# B&R Automation Studio project BottleFiller (part 2)

#### Main.st
```iecst
PROGRAM _INIT
	(* Insert code here *)
	//Conveyor parameters
	MpAxisConvParType.AutoTune.Mode:=mcAXIS_TUNE_AUTOMATIC;
	MpAxisConvParType.AutoTune.MaxCurrentPercent:=80;
	MpAxisConvParType.AutoTune.MaxDistance:=30;
	MpAxisConvParType.AutoTune.MaxPositionError:=30;
	//Nozzle parameters
	MpAxisNozzleParType := MpAxisConvParType;
	MpAxisNozzleParType.Homing.Position:=195;
	//Cart parameters
	MpAxisCartParType := MpAxisConvParType;

	camNozzleParameters.CamSequence.Get.GetOnEnable:=1;
	camNozzleParameters.CamSequence.Get.Command:=mcGET_PAR_ACTUAL;
	camNozzleParameters.CamSequence.Data.DataAddress:=ADR(configCamNozzle);
	camNozzleParameters.CamSequence.Data.DataSize:=SIZEOF(configCamNozzle);
	camNozzleParameters.CamSequence.Set.Command:=mcSET_UPDATE_FROM_ADR;
	camNozzleParameters.CamSequence.Set.Mode:=mcAXIS_CAM_SEQ_SET_ON_UPDATE;
END_PROGRAM

PROGRAM _CYCLIC
	(* Insert code here *)
	//axis declaration
	MpAxisConv(MpLink := ADR(axisConv), Enable := 1, Parameters := ADR(MpAxisConvParType), AutoTune := 1);
	MpAxisCart(MpLink := ADR(axisCart), Enable := 1, Parameters := ADR(MpAxisCartParType),   AutoTune := 1);
	MpAxisNozzle(MpLink := ADR(axisNozzle), Enable := 1, Parameters := ADR(MpAxisNozzleParType),  AutoTune := 1);

	//sequence parameters
	configCamNozzle.State[3].CamID:=STRING_TO_USINT(gControl.currentBottleType);

	//Sequence declaration
	camSeq(MpLink := ADR(axisCart), Enable := 1, Parameters := ADR(camParameters), MpLinkMaster := ADR(axisConv));
	camSeqNozzle(MpLink := ADR(axisNozzle), Enable := 1, Parameters := ADR(camNozzleParameters), MpLinkMaster := ADR(axisConv));

	//conveyor management
	MpAxisConvParType.Velocity:=gAxisUpdate.Conveyor.Velocity;
	MpAxisConv.ErrorReset:=gControl.Conveyor.errorReset;
	MpAxisConv.Power:=gControl.power;
	MpAxisConv.Home:=gControl.Conveyor.home;
	MpAxisConv.Stop:=gControl.Conveyor.stop;
	MpAxisConv.JogNegative:=gControl.Conveyor.jogNegative;
	MpAxisConv.JogPositive:=gControl.Conveyor.jogPositive;

	//Cart management
	MpAxisCart.ErrorReset:=gControl.Cart.errorReset;
	MpAxisCart.Power:=gControl.power;
	MpAxisCart.Home:=gControl.Cart.home;
	MpAxisCart.Stop:=gControl.Cart.stop;
	MpAxisCart.JogNegative:=gControl.Cart.jogNegative;
	MpAxisCart.JogPositive:=gControl.Cart.jogPositive;

	//nozzle Management
	MpAxisNozzle.ErrorReset:=gControl.Nozzle.errorReset;
	MpAxisNozzle.Power:=gControl.power;
	MpAxisNozzle.Home:=gControl.Nozzle.home;
	MpAxisNozzle.Stop:=gControl.Nozzle.stop;
	MpAxisNozzle.JogNegative:=gControl.Nozzle.jogNegative;
	MpAxisNozzle.JogPositive:=gControl.Nozzle.jogPositive;

	//cam params
//	camSeq.Signal1:=gCamSeqParam.cart.signal1;
	camSeqNozzle.Signal1:=gCamSeqParam.nozzle.signal1;

	IF camSeqNozzle.UpdateDone THEN
		camSeqNozzle.Update:=0;
	END_IF;
	IF MpAxisConv.UpdateDone THEN
		MpAxisConv.Update:=0;
	END_IF;
	IF MpAxisNozzle.UpdateDone THEN
		MpAxisNozzle.Update:=0;
	END_IF;
	IF MpAxisCart.UpdateDone THEN
		MpAxisCart.Update:=0;
	END_IF;

	IF gControl.needUpdate THEN

		//conveyor
		MpAxisConvParType.Velocity:=STRING_TO_UINT(gAxisUpdate.staticVelocity);
		MpAxisConvParType.Jog.LimitPosition.FirstPosition:=gAxisUpdate.Conveyor.FirstPosition;
		MpAxisConvParType.Jog.LimitPosition.LastPosition:=gAxisUpdate.Conveyor.LastPosition;
		MpAxisConvParType.Position:=gAxisUpdate.Conveyor.Position;
		//MpAxisConvParType.Homing.Mode:=gAxisUpdate.Conveyor.Homing;
		//MpAxisConvParType.Velocity:=gAxisUpdate.Conveyor.Velocity;
		MpAxisConvParType.Jog.Velocity:=gAxisUpdate.Conveyor.Velocity;

		//cart
		MpAxisCartParType.Jog.LimitPosition.FirstPosition:=gAxisUpdate.Cart.FirstPosition;
		MpAxisCartParType.Jog.LimitPosition.LastPosition:=gAxisUpdate.Cart.LastPosition;
		MpAxisCartParType.Position:=gAxisUpdate.Cart.Position;
		//	MpAxisCartParType.Homing.Mode:=gAxisUpdate.Cart.Homing;
		MpAxisCartParType.Jog.Velocity:=50;

		//nozzle
		MpAxisNozzleParType.Jog.LimitPosition.FirstPosition:=gAxisUpdate.Nozzle.FirstPosition;
		MpAxisNozzleParType.Jog.LimitPosition.LastPosition:=gAxisUpdate.Nozzle.LastPosition;
		MpAxisNozzleParType.Position:=gAxisUpdate.Nozzle.Position;
		//	MpAxisNozzleParType.Homing.Mode:=gAxisUpdate.Nozzle.Homing;
		MpAxisNozzleParType.Jog.Velocity:=50;

		MpAxisNozzle.Update:=1;
		MpAxisConv.Update:=1;
		MpAxisCart.Update:=1;

		IF MpAxisNozzle.UpdateDone THEN
			MpAxisNozzle.Update:=0;
		END_IF;
		IF MpAxisCart.UpdateDone THEN
			MpAxisCart.Update:=0;
		END_IF;
		IF MpAxisConv.UpdateDone THEN
			MpAxisConv.Update:=0;
		END_IF;
		gControl.needUpdate:=0;
	END_IF;

	CASE gAxisCase OF
		HOLDON:
			IF NOT (MpAxisCart.Stopped AND MpAxisConv.Stopped AND MpAxisNozzle.Stopped)  THEN
				MpAxisCart.Stop:=1;
				MpAxisConv.Stop:=1;
				MpAxisNozzle.Stop:=1;
			END_IF;

			IF  MpAxisConv.Info.PLCopenState = mcAXIS_STANDSTILL AND MpAxisCart.Info.PLCopenState = mcAXIS_STANDSTILL AND MpAxisNozzle.Info.PLCopenState = mcAXIS_STANDSTILL THEN
				MpAxisCart.Stop:=0;
				MpAxisConv.Stop:=0;
				MpAxisNozzle.Stop:=0;
				gMainAction.stopped:=1;
			END_IF;

		POWERED:
			IF (gControl.power AND NOT gControl.stop AND NOT gAxisOutputs.Conveyor.error) THEN //error
				//power on axis
				MpAxisCart.Power:=1;
				MpAxisConv.Power:=1;
				MpAxisNozzle.Power:=1;

				IF MpAxisCart.PowerOn AND MpAxisConv.PowerOn AND MpAxisNozzle.PowerOn THEN
					gMainAction.powered:=1;
				END_IF;

			END_IF;

		HOMING:
			gControl.bottleCnt:=0;
			MpAxisCart.Home:=1;
			MpAxisConv.Home:=1;
			MpAxisNozzle.Home:=1;
			gMainAction.homed:=1;

		STANDSTILL:
			IF gControl.start THEN
				IF gControl.manual THEN
					gAxisCase:=onMOVE;
				ELSE
					gAxisCase:=CONNECT;
				END_IF;
			END_IF;

		CONNECT:
			MpAxisCart.Home:=0;
			MpAxisConv.Home:=0;
			MpAxisNozzle.Home:=0;
			camSeq.EndSequence:=0;
			camSeqNozzle.EndSequence:=0;
			camSeq.ErrorReset:=0;
			camSeq.StartSequence:=1;
			camSeqNozzle.StartSequence:=1;

			IF camSeq.Error THEN
				camSeq.ErrorReset:=1;
				camSeq.StartSequence:=0;
			END_IF;

			IF camSeq.InCam AND camSeqNozzle.InCam THEN
				camSeq.Signal1:=1;
				gMainAction.connected:=1;
				connectHelper:=0;
			END_IF;

		DISCONNECT:
			MpAxisCart.Home:=0;
			MpAxisConv.Home:=0;
			MpAxisNozzle.Home:=0;
			gMainAction.connected:=0;
			MpAxisConv.MoveVelocity:=0;
			camSeq.Signal1:=0;
			camSeqNozzle.Signal1:=0;
			camSeq.StartSequence:=0;
			camSeq.EndSequence:=1;
			camSeqNozzle.StartSequence:=0;
			camSeqNozzle.EndSequence:=1;
			IF NOT (camSeq.Running AND camSeqNozzle.Running) THEN
				gMainAction.disconnected:=1;
			END_IF;

		onMOVE:
			//karetka
			IF mouseEvent THEN
				IF gControl.Cart.safeLevelStop THEN
					gControl.Cart.stop:=gControl.Cart.safeLevelStop;
					IF MpAxisCartParType.Direction = 1 AND MpAxisCart.Position >= gControl.Cart.upperLimit THEN
						gControl.Cart.safeLevelStop:=0;
						gControl.Cart.stop:=0;
					ELSIF MpAxisCartParType.Direction = 0 AND MpAxisCart.Position <= gControl.Cart.lowerLimit THEN
						gControl.Cart.safeLevelStop:=0;
						gControl.Cart.stop:=0;
					END_IF;
				END_IF;

				IF gControl.Nozzle.safeLevelStop THEN
					gControl.Nozzle.stop:=gControl.Nozzle.safeLevelStop;
					IF MpAxisNozzleParType.Direction = 1 AND MpAxisNozzle.Position >= gControl.Nozzle.upperLimit THEN
						gControl.Nozzle.safeLevelStop:=0;
						gControl.Nozzle.stop:=0;
					ELSIF MpAxisNozzleParType.Direction = 0 AND MpAxisNozzle.Position <= gControl.Nozzle.lowerLimit THEN
						gControl.Nozzle.safeLevelStop:=0;
						gControl.Nozzle.stop:=0;
					END_IF;
				END_IF;

				MpAxisConv.MoveVelocity:=gControl.moveVelocity;

				IF gControl.Cart.onlyRight AND MpAxisCartParType.Direction = 0 THEN
					gControl.Cart.stop:=0;
					MpAxisCart.MoveVelocity:=gControl.Cart.moveVelocity;
				END_IF;

				IF gControl.Cart.onlyLeft AND MpAxisCartParType.Direction = 1 THEN
					gControl.Cart.stop:=0;
					MpAxisCart.MoveVelocity:=gControl.Cart.moveVelocity;
				END_IF;

				IF NOT gControl.Cart.onlyLeft AND NOT gControl.Cart.onlyRight THEN
					MpAxisCart.MoveVelocity:= NOT gControl.Cart.safeLevelStop AND gControl.Cart.moveVelocity;
				END_IF;

				//nozzle
				IF gControl.Nozzle.onlyRight AND MpAxisNozzleParType.Direction = 0 THEN
					gControl.Nozzle.stop:=0;
					MpAxisNozzle.MoveVelocity:=gControl.Nozzle.moveVelocity;
				END_IF;

				IF gControl.Nozzle.onlyLeft AND MpAxisNozzleParType.Direction = 1 THEN
					gControl.Nozzle.stop:=0;
					MpAxisNozzle.MoveVelocity:=gControl.Nozzle.moveVelocity;
				END_IF;

				IF NOT gControl.Nozzle.onlyLeft AND NOT gControl.Nozzle.onlyRight THEN
					MpAxisNozzle.MoveVelocity:= NOT gControl.Nozzle.safeLevelStop AND gControl.Nozzle.moveVelocity;
				END_IF;
			ELSE
				MpAxisConv.MoveVelocity:=gControl.moveVelocity;
				MpAxisConv.JogNegative:=gControl.Conveyor.jogNegative;
				MpAxisConv.JogPositive:=gControl.Conveyor.jogPositive;
				MpAxisCart.JogNegative:=gControl.Cart.jogNegative;
				MpAxisCart.JogPositive:=gControl.Cart.jogPositive;
				MpAxisNozzle.JogNegative:=gControl.Nozzle.jogNegative;
				MpAxisNozzle.JogPositive:=gControl.Nozzle.jogPositive;
			END_IF;
			IF MpAxisConv.Position > 0 THEN
				gMainAction.homed:=0;
			END_IF;

	END_CASE;

	controlInfo.Conveyor.error:=MpAxisConv.Error;
	controlInfo.Conveyor.isHomed:=MpAxisConv.IsHomed;
	controlInfo.Conveyor.isPowered:=MpAxisConv.PowerOn;
	controlInfo.Conveyor.position:=LREAL_TO_REAL(MpAxisConv.Position);
	controlInfo.Conveyor.velocity:=MpAxisConv.Velocity;
	controlInfo.Conveyor.updateDone:=MpAxisConv.UpdateDone;
	controlInfo.Conveyor.MoveActive:=MpAxisConv.Info.Jogging;

	controlInfo.Cart.error:=MpAxisCart.Error;
	controlInfo.Cart.isHomed:=MpAxisCart.IsHomed;
	controlInfo.Cart.isPowered:=MpAxisCart.PowerOn;
	controlInfo.Cart.position:=LREAL_TO_REAL(MpAxisCart.Position);
	controlInfo.Cart.velocity:=MpAxisCart.Velocity;
	controlInfo.Cart.updateDone:=MpAxisCart.UpdateDone;
	controlInfo.Cart.MoveActive:=MpAxisCart.Info.Jogging;

	controlInfo.Nozzle.error:=MpAxisNozzle.Error;
	controlInfo.Nozzle.isHomed:=MpAxisNozzle.IsHomed;
	controlInfo.Nozzle.isPowered:=MpAxisNozzle.PowerOn;
	controlInfo.Nozzle.position:=LREAL_TO_REAL(MpAxisNozzle.Position);
	controlInfo.Nozzle.velocity:=MpAxisNozzle.Velocity;
	controlInfo.Nozzle.updateDone:=MpAxisNozzle.UpdateDone;
	controlInfo.Nozzle.MoveActive:=MpAxisNozzle.Info.Jogging;

	gCamSeqParam.cart.currentStateIndex:=camSeq.ActualStateIndex;
	gCamSeqParam.nozzle.currentStateIndex:=camSeq.ActualStateIndex;

	gAxisOutputs:=controlInfo;

END_PROGRAM

PROGRAM _EXIT
	(* Insert code here *)

END_PROGRAM
```

### Program Logical/Simulation/Logic/BottleFiller

#### Types.typ
```iecst
TYPE
	SimulationAxisPositionEnum : 	STRUCT
		Conveyor : REAL;
		Cart : REAL;
		Nozzle : REAL;
	END_STRUCT;
	bottleFillerRecipeEnum : 	STRUCT
		diPumpSpeedFlow : INT := 0;
		diVelocity : REAL := 0.0;
		diSpeedProfile : INT := 0;
		diBottleShape : INT := 0;
	END_STRUCT;
	FillerEnum :
		( (*Every possible case*)
		DISABLED,
		STOP,
		SERVICE,
		INIT,
		AUTOMAT,
		ERROR
		);
END_TYPE
```

#### Variables.var
```iecst
(*case machine*)
VAR
	FillerTyp : FillerEnum;
	bottleFillerRecipeTyp : bottleFillerRecipeEnum;
END_VAR
(*digital inputs*)
VAR
	diError : BOOL;
	diManual : BOOL := FALSE; (*Determine if machine works automatically or needs manual control*)
	diStop : BOOL := FALSE; (*Stop switch*)
	diStart : BOOL := FALSE; (*Start switch*)
	diPowerSwitch : BOOL := FALSE; (*Power on switch*)
	diLiquidLevel : REAL := 100;
	diConveyorHomingSwitch : BOOL := FALSE; (*Sensor detecting conveyor at homing position*)
	diNozzleHomingSwitch : BOOL := FALSE; (*Sensor detecting nozzle at homing position*)
	diCartHomingSwitch : BOOL := FALSE; (*Sensor detecting cart at homing position*)
	diBottleDetection : BOOL := FALSE; (*Sensor detecting presence of a bottle*)
END_VAR
(*digital outputs*)
VAR
	doPumpRelay : INT; (*Output controlling the pump building pressure for liquid flow*)
	doValveRelay : BOOL; (*Output controlling the liquid valve opening*)
END_VAR
(*analog outputs*)
VAR
	aoPumpFlowSpeed : ARRAY[0..100] OF INT; (*Datapoint in percentage to the pump system about liquid flow speed in percent*)
END_VAR
(*other variables*)
VAR
	roleInfo : MpUserXMgrUIRoleInfoType;
	MpBFRecipeXml : MpRecipeXml;
	MpBFRecipeRegPar : MpRecipeRegPar; (*MpBFRecipeHMI : MpRecipeUI;
	UISetup : MpRecipeUISetupType;
	MpRecipeUIConnectType : MpRecipeUIConnectType;*)
	MpAxisConvParType : MpAxisBasicParType;
	camSeq : MpAxisCamSequencer;
	inCam : BOOL;
	camSeqNozzle : MpAxisCamSequencer;
	camParameters : MpAxisCamSequencerParType;
	MpAxisConv : MpAxisBasic;
	MpAxisCart : MpAxisBasic;
	MpAxisNozzle : MpAxisBasic;
	SimulationAxisPosition : SimulationAxisPositionEnum;
	changedPosition : BOOL;
	MpAxisCartParType : MpAxisBasicParType;
	MpAxisNozzleParType : MpAxisBasicParType;
END_VAR
```

#### Main.st
```iecst
PROGRAM _INIT
	(* Insert code here *)
	 FillerTyp:=DISABLED;
END_PROGRAM

PROGRAM _CYCLIC
	(* Insert code here *)
//	MpBFRecipeXml(MpLink := ADR(BFRecipe) , Enable := 1, DeviceName := ADR('USER') , FileName := ADR('BottleFillerRecipe'));
//	MpBFRecipeRegPar(MpLink := ADR(BFRecipe), Enable := 1, PVName := ADR('BootleFiller:bottleFillerRecipeTyp'));
//	MpBFRecipeHMI(MpLink := ADR(BFRecipe), Enable := 1 , ErrorReset := , UISetup := ADR(UISetup) , UIConnect := ADR(MpRecipeUIConnectType));
	MpAxisConvParType.AutoTune.Mode:=mcAXIS_TUNE_AUTOMATIC;
	MpAxisConvParType.AutoTune.MaxCurrentPercent:=80;
	MpAxisConvParType.AutoTune.MaxDistance:=30;
	MpAxisConvParType.AutoTune.MaxPositionError:=30;
	MpAxisNozzleParType.Homing.Position:=200;
	MpAxisConv(MpLink := ADR(axisConv), Enable := 1, Parameters := ADR(MpAxisConvParType), AutoTune := 1);
	MpAxisCart(MpLink := ADR(axisCart), Enable := 1, Parameters := ADR(MpAxisCartParType),   AutoTune := 1);
	MpAxisNozzle(MpLink := ADR(axisNozzle), Enable := 1, Parameters := ADR(MpAxisNozzleParType),  AutoTune := 1);

//
//	MpBFRecipeXml();

	camSeq(MpLink := ADR(axisCart), Enable := 1, Parameters := ADR(camParameters), MpLinkMaster := ADR(axisConv));
	camSeqNozzle(MpLink := ADR(axisNozzle), Enable := 1, Parameters := ADR(camParameters), MpLinkMaster := ADR(axisConv));

	SimulationAxisPosition.Cart := LREAL_TO_REAL(MpAxisCart.Position);
	SimulationAxisPosition.Conveyor := LREAL_TO_REAL(MpAxisConv.Position);
	SimulationAxisPosition.Nozzle := LREAL_TO_REAL(MpAxisNozzle.Position);
	gAdrAxesPositions := ADR(SimulationAxisPosition);
	//MpBFRecipeHMI();
	CASE FillerTyp OF
		DISABLED:
			diStart:=0;
			diStop:=0;

			IF diPowerSwitch THEN
				FillerTyp:=INIT;
			END_IF;

		INIT:
			//procedury początkowe; home, kierunek
			IF diPowerSwitch AND NOT diStop AND NOT diError THEN

				//power on axis
				MpAxisCart.Power:=1;
				MpAxisConv.Power:=1;
				MpAxisNozzle.Power:=1;

				//homing
				MpAxisCart.Home:=1;
				IF MpAxisCart.IsHomed THEN
					MpAxisCart.Home:=0;
				END_IF;

				MpAxisConv.Home:=1;
				IF MpAxisConv.IsHomed THEN
					MpAxisConv.Home:=0;
				END_IF;

				MpAxisNozzle.Home:=1;
				IF MpAxisNozzle.IsHomed THEN
					MpAxisNozzle.Home:=0;
				END_IF;

				IF diStart AND MpAxisNozzle.IsHomed AND MpAxisConv.IsHomed AND MpAxisCart.IsHomed AND MpAxisCart.PowerOn AND MpAxisNozzle.PowerOn AND MpAxisConv.PowerOn THEN
					//power on camSeq

					IF diManual THEN
						FillerTyp:=SERVICE;
					ELSE
						camSeq.StartSequence:=1;
						camSeqNozzle.StartSequence:=1;
						FillerTyp:= AUTOMAT;
					END_IF;
				END_IF;
			END_IF;

		AUTOMAT:
			IF camSeq.InCam AND camSeqNozzle.InCam THEN

				camSeq.Signal1:=1;
				camSeqNozzle.Signal1:=1;
				MpAxisConv.MoveVelocity := (diStart AND NOT diStop);
				IF MpAxisConv.UpdateDone THEN
					MpAxisConv.Update:=0;
				END_IF;

			END_IF;

		SERVICE:
			//odpalenie cam-ów
			IF inCam THEN
				IF changedPosition THEN

					MpAxisCartParType.Homing.Mode:=141;
					MpAxisCartParType.Homing.Options.HomingVelocity:=50;
					MpAxisCart.Update:=1;

					MpAxisConvParType.Homing.Mode:=141;
					MpAxisConvParType.Homing.Options.HomingVelocity:=50;
					MpAxisConv.Update:=1;

					MpAxisNozzleParType.Homing.Mode:=141;
					MpAxisNozzleParType.Homing.Options.HomingVelocity:=50;
					MpAxisNozzle.Update:=1;

					IF MpAxisCart.UpdateDone THEN
						MpAxisCart.Home:=1;
						MpAxisCart.Update:=0;
					END_IF;
					IF MpAxisConv.UpdateDone THEN
						MpAxisConv.Home:=1;

						MpAxisConv.Update:=0;
					END_IF;
					IF MpAxisNozzle.UpdateDone THEN
						MpAxisNozzle.Home:=1;

						MpAxisNozzle.Update:=0;
					END_IF;
					changedPosition:=0;
				END_IF;

				IF camSeq.InCam AND camSeqNozzle.InCam THEN
					camSeq.Signal1:=1;
					camSeqNozzle.Signal1:=1;
				END_IF;

				IF camSeq.Signal1 AND camSeqNozzle.Signal1 THEN

					IF MpAxisConv.InPosition THEN
						MpAxisConv.MoveAbsolute:=0;
						MpAxisConv.MoveAdditive:=0;
						MpAxisConv.MoveVelocity:=0;
					END_IF;
					//switch update taśmy

					IF MpAxisConv.UpdateDone THEN
						MpAxisConv.Update:=0;
					END_IF;
				END_IF;

			END_IF;

			//wyłączenie cam-ów
			IF EDGENEG(inCam) THEN
				camSeq.StartSequence:=0;
				camSeqNozzle.StartSequence:=0;
				camSeq.Signal1:=0;
				camSeqNozzle.Signal1:=0;
			END_IF;

			//obsługa zmiany kierunków ruchu urządzeń przy obsłudze manualnej
			IF EDGEPOS(MpAxisConv.MoveAbsolute) THEN
				IF MpAxisConv.Position > MpAxisConvParType.Position THEN
					MpAxisConvParType.Direction:=mcDIR_NEGATIVE;
					MpAxisConv.Update:=1;
				ELSIF MpAxisConv.Position < MpAxisConvParType.Position THEN
					MpAxisConvParType.Direction:=mcDIR_POSITIVE;
					MpAxisConv.Update:=1;
				END_IF;
			END_IF;

			//wyłączanie ruchu taśmy
			IF MpAxisConv.Info.JogLimitReached THEN
				MpAxisConv.JogNegative:=0;
				MpAxisConv.JogPositive:=0;
			END_IF;
			//switch update taśmy
			IF MpAxisConv.UpdateDone THEN
				MpAxisConv.Update:=0;
			END_IF;

			//wyłączanie jog-ów karetki po dojechaniu na miejsce
			IF MpAxisCart.Info.JogLimitReached THEN
				MpAxisCart.JogNegative:=0;
				MpAxisCart.JogPositive:=0;
			END_IF;
			//switch update karetki
			IF MpAxisCart.UpdateDone THEN
				MpAxisCart.Update:=0;
			END_IF;

			//wyłączanie jog-ów dyszy po dojechaniu na miejsce
			IF MpAxisNozzle.Info.JogLimitReached THEN
				MpAxisNozzle.JogNegative:=0;
				MpAxisNozzle.JogPositive:=0;
			END_IF;
			//switch update karetki
			IF MpAxisNozzle.UpdateDone THEN
				MpAxisNozzle.Update:=0;
			END_IF;

			IF NOT diManual THEN
				FillerTyp:=AUTOMAT;
			END_IF;

		ERROR:

		STOP:

	END_CASE;

END_PROGRAM

PROGRAM _EXIT
	(* Insert code here *)

END_PROGRAM
```

### Types.typ
```iecst
TYPE
	bottleFillerRecipeEnum : 	STRUCT
		diPumpSpeedFlow : USINT := 0;
		diVelocity : USINT := 0;
		diSpeedProfile : USINT := 0;
		diBottleShape : USINT := 0;
	END_STRUCT;
	FillerEnum :
		( (*Every possible case*)
		DISABLED,
		STOP,
		SERVICE,
		INIT,
		AUTOMAT,
		ERROR
	);
END_TYPE
```

### Variables.var
```iecst
(*case machine*)
VAR
	FillerTyp : FillerEnum;
	bottleFillerRecipeTyp : bottleFillerRecipeEnum;
END_VAR
(*digital inputs*)
VAR
	diConveyorHomingSwitch : BOOL := FALSE; (*Sensor detecting conveyor at homing position*)
	diNozzleHomingSwitch : BOOL := FALSE; (*Sensor detecting nozzle at homing position*)
	diCartHomingSwitch : BOOL := FALSE; (*Sensor detecting cart at homing position*)
	diBottleDetection : BOOL := FALSE; (*Sensor detecting presence of a bottle*)
END_VAR
(*digital outputs*)
VAR
	doPumpRelay : BOOL; (*Output controlling the pump building pressure for liquid flow*)
	doValveRelay : BOOL; (*Output controlling the liquid valve opening*)
END_VAR
(*analog outputs*)
VAR
	aoPumpFlowSpeed : ARRAY[0..100] OF INT; (*Datapoint in percentage to the pump system about liquid flow speed in percent*)
END_VAR
(*other variables*)
VAR
	roleInfo : MpUserXMgrUIRoleInfoType;
	MpBFRecipeXml : MpRecipeXml;
	MpBFRecipeRegPar : MpRecipeRegPar;
	(*MpBFRecipeHMI : MpRecipeUI;
	UISetup : MpRecipeUISetupType;
	MpRecipeUIConnectType : MpRecipeUIConnectType;*)
END_VAR
```

Listed in the project but not available here: Logical/Global.typ, Logical/BottleFiller/workTasks/GlobalRobVis.var, Logical/BottleFiller/workTasks/RobVis, Logical/BottleFiller/workTasks/Simulation, Logical/Package/Variables1.var, Logical/Simulation/Logic/GlobalRobVis.typ, Logical/Simulation/Sim
